TYPE AX5000_S_0047 :
STRUCT
	Position_command_valut:DINT;
END_STRUCT
END_TYPE

(* stored: Version 1.1.0.1, ProductVersion 3.1.4024.3
   DUT AX5000_S_0047: Id {51ca9d8f-69a3-4d1c-8f25-e13d528f852c} *)
